(* CODESYS project Lib_DebugLogger_01.library
   Author: Aliazzzz
   Version: 0.0.0.1
   Description: Reworked by Aliazzzz
      
      Original library by Sebastian Rau
   Title: DebugLogger
   DefaultNamespace: DebugLogger
   Company: Aliazzzz

Project tree, tasks and I/O mapping:
  Data types/
    data type E_DebugMessagePriority
    data type ST_DEBUG
    data type ST_DEBUG_MESSAGE
  Library Information/
    function GetLibVersion [ST]
    function GetLibVersionNumber [ST]
    function IsLibReleased [ST]
  POUs/
    function DebugLog [ST]
  global variables GVL_DEBUG
  global variables DebugLogParam
*)

// Data types/E_DebugMessagePriority
TYPE E_DebugMessagePriority :
(
	DEBUG 	:= 0,
	INFO 	:= 1,
	WARN 	:= 2,
	ERROR 	:= 3,
	FATAL 	:= 4
);
END_TYPE

// Data types/ST_DEBUG
TYPE ST_DEBUG :
STRUCT
	(* aMessages : ARRAY[0..GVL_DEBUG.iMaxDebugEntries] OF ST_DEBUG_MESSAGE; *)
	aMessages : ARRAY[0..DebugLogParam.iMaxDebugEntries] OF ST_DEBUG_MESSAGE;
	iIndex : INT;
	eMinLogPriority : E_DebugMessagePriority := DEBUG;
	dtActualTime : DT;  (* Results in *NOW* *)
END_STRUCT
END_TYPE

// Data types/ST_DEBUG_MESSAGE
TYPE ST_DEBUG_MESSAGE :
STRUCT
	tTime		: DT;
	sMessage 	: STRING(64);
	ePriority	: E_DebugMessagePriority;
END_STRUCT
END_TYPE

// GVL_DEBUG
VAR_GLOBAL
	stDebugInformation : ST_DEBUG;
END_VAR

(*
VAR_GLOBAL CONSTANT
	iMaxDebugEntries : INT := 128;
END_VAR
*)

// DebugLogParam
{attribute 'qualified_only'}
VAR_GLOBAL CONSTANT
	iMaxDebugEntries : INT := 128;
END_VAR

// Library Information/GetLibVersion
// This function has been automatically generated from the project information.
FUNCTION GetLibVersion : VERSION
VAR_INPUT
	
END_VAR

GetLibVersion.uiMajor := 0;
GetLibVersion.uiMinor := 0;
GetLibVersion.uiServicePack := 0;
GetLibVersion.uiPatch := 1;

END_FUNCTION

// POUs/DebugLog
FUNCTION DebugLog : BOOL
VAR_INPUT
	sMessage 	: STRING(64);
	ePriority 	: E_DebugMessagePriority;
END_VAR

IF ePriority >=  stDebugInformation.eMinLogPriority THEN
	
	stDebugInformation.aMessages[stDebugInformation.iIndex].sMessage := sMessage;
	stDebugInformation.aMessages[stDebugInformation.iIndex].tTime := stDebugInformation.dtActualTime;
	stDebugInformation.aMessages[stDebugInformation.iIndex].ePriority := ePriority;

	(*IF stDebugInformation.iIndex < iMaxDebugEntries THEN*)
	IF stDebugInformation.iIndex < debuglogparam.iMaxDebugEntries THEN

		stDebugInformation.iIndex := stDebugInformation.iIndex +1;
	ELSE
		stDebugInformation.iIndex := 0;
	END_IF
	
	DebugLog := TRUE;
ELSE
	DebugLog := FALSE;
END_IF

END_FUNCTION

// Library Information/GetLibVersionNumber
// This function has been automatically generated from the project information.
FUNCTION GetLibVersionNumber : DWORD
VAR_INPUT
	
END_VAR

GetLibVersionNumber := 1;

END_FUNCTION

// Library Information/IsLibReleased
// This function has been automatically generated from the project information.
FUNCTION IsLibReleased : BOOL
VAR_INPUT
	
END_VAR

IsLibReleased := FALSE;

END_FUNCTION
